// Mitsubishi GX Works2 project: Uni-CVX300R   PLC: FX3S

PROGRAM MAIN
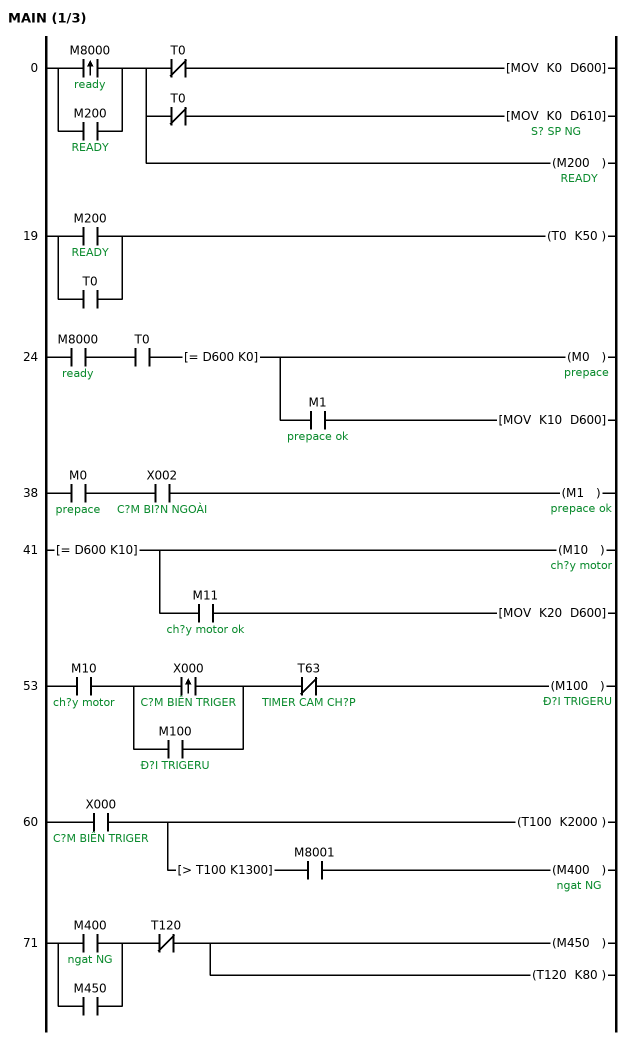
0     LDP     M8000  ; ready
      OR      M200  ; READY
      MPS
      ANI     T0
      MOV     K0 D600
      MRD
      ANI     T0
      MOV     K0 D610  ; S? SP NG
      MPP
      OUT     M200  ; READY
19    LD      M200  ; READY
      OR      T0
      OUT     T0 K50
24    LD      M8000  ; ready
      AND     T0
      AND=    D600 K0
      OUT     M0  ; prepace
      AND     M1  ; prepace ok
      MOV     K10 D600
38    LD      M0  ; prepace
      AND     X002  ; C?M BI?N NGOÀI
      OUT     M1  ; prepace ok
41    LD=     D600 K10
      OUT     M10  ; ch?y motor
      AND     M11  ; ch?y motor ok
      MOV     K20 D600
53    LD      M10  ; ch?y motor
      LDP     X000  ; C?M BIÊN TRIGER
      OR      M100  ; Ð?I TRIGERU
      ANB
      ANI     T63  ; TIMER CAM CH?P
      OUT     M100  ; Ð?I TRIGERU
60    LD      X000  ; C?M BIÊN TRIGER
      OUT     T100 K2000
      AND>    T100 K1300
      AND     M8001
      OUT     M400  ; ngat NG
71    LD      M400  ; ngat NG
      OR      M450
      ANI     T120
      OUT     M450
      OUT     T120 K80
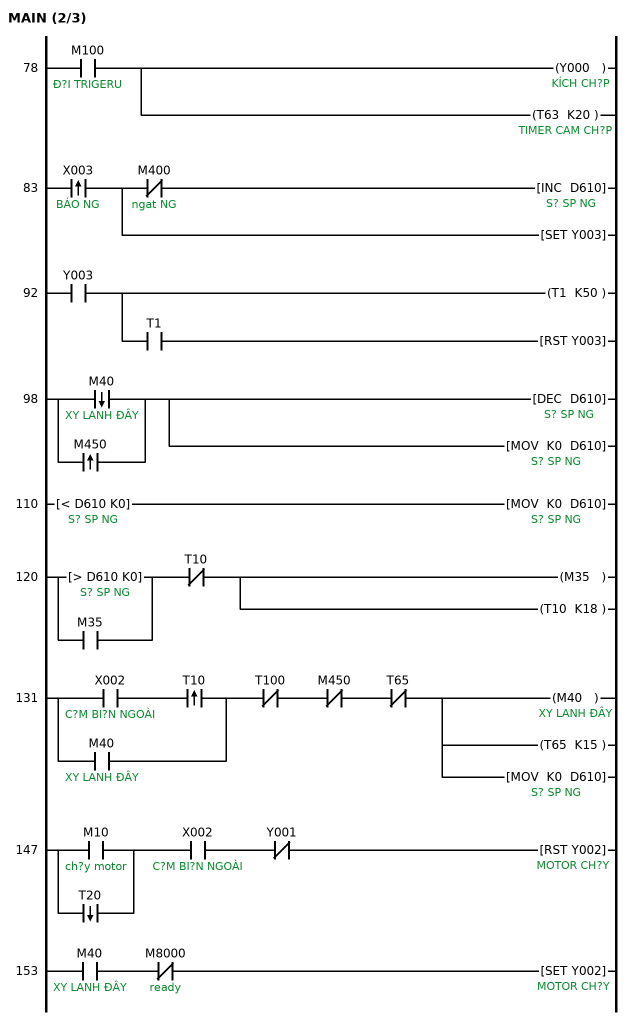
78    LD      M100  ; Ð?I TRIGERU
      OUT     Y000  ; KÍCH CH?P
      OUT     T63 K20  ; TIMER CAM CH?P
83    LDP     X003  ; BÁO NG
      MPS
      ANI     M400  ; ngat NG
      INC     D610
      MPP
      SET     Y003
92    LD      Y003
      OUT     T1 K50
      AND     T1
      RST     Y003
98    LDF     M40  ; XY LANH ÐÂY
      ORP     M450
      DEC     D610
      MOV     K0 D610
110   LD<     D610 K0  ; S? SP NG
      MOV     K0 D610
120   LD>     D610 K0  ; S? SP NG
      OR      M35
      ANI     T10
      OUT     M35
      OUT     T10 K18
131   LD      X002  ; C?M BI?N NGOÀI
      ANDP    T10
      OR      M40  ; XY LANH ÐÂY
      ANI     T100
      ANI     M450
      ANI     T65
      OUT     M40  ; XY LANH ÐÂY
      OUT     T65 K15
      MOV     K0 D610
147   LD      M10  ; ch?y motor
      ORF     T20
      AND     X002  ; C?M BI?N NGOÀI
      ANI     Y001
      RST     Y002  ; MOTOR CH?Y
153   LD      M40  ; XY LANH ÐÂY
      ANI     M8000  ; ready
      SET     Y002  ; MOTOR CH?Y
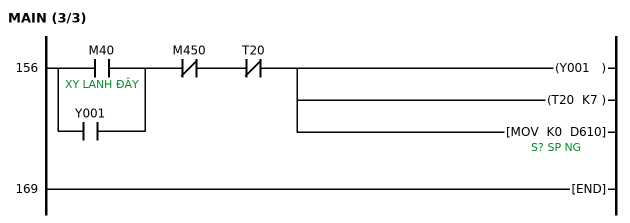
156   LD      M40  ; XY LANH ÐÂY
      OR      Y001
      ANI     M450
      ANI     T20
      OUT     Y001
      OUT     T20 K7
      MOV     K0 D610
169   END
END_PROGRAM

// device comments not shown above
M15  ; Ð?I CAMARA CH?P
M16  ; Ð?I OK
M20  ; camera check
M21  ; CHECK CAMERA OK
M25  ; CAMERA TR? V?
M26  ; CAMERA TR? V? NG
M30  ; BANG T?I D?NG
M31  ; BANG T?I D?NG OK
M41  ; XY LANH ÐÂY OK
M101  ; XY LANH ÐAY]
X001  ; C?M BI?N XY LANH
Y004  ; Báo L?i
T30  ; DELAY XY LANH TH
